% RSLogix 500 project aula1.RSS, saved by version 8.30.00.16 %
PROJECT "UNTITLED"    % processor: Bul.1763 MicroLogix 1100 Series B %

PROGRAM FILES
  LAD 2   6 rungs

DATA FILES
  O0 OUTPUT  4 elements
  I1 INPUT  6 elements
  S2 STATUS  66 elements
  B3 BINARY  1 elements
  T4 TIMER  1 elements
  C5 COUNTER  1 elements
  R6 CONTROL  1 elements
  N7 INTEGER  1 elements
  F8 FLOAT  1 elements

LADDER 2
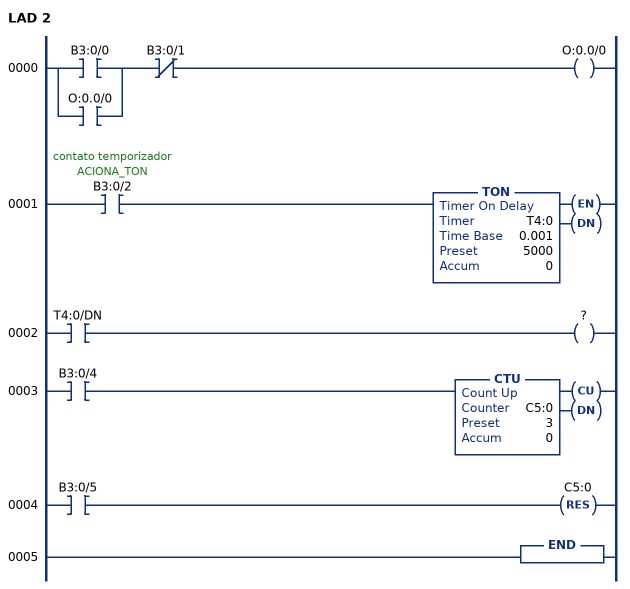
% Rung: 0 %
SOR BST XIC B3:0/0 NXB XIC O:0.0/0 BND XIO B3:0/1 OTE O:0.0/0 EOR
% Rung: 1 %  % edit flag set %
SOR XIC B3:0/2 TON T4:0 0.001 5000 0 EOR
%   B3:0/2  ACIONA_TON  "contato temporizador" %
% Rung: 2 %  % edit flag set %
SOR XIC T4:0/DN OTE ? EOR
% Rung: 3 %  % edit flag set %
SOR XIC B3:0/4 CTU C5:0 3 0 EOR
% Rung: 4 %  % edit flag set %
SOR XIC B3:0/5 RES C5:0 EOR
% Rung: 5 %
SOR END EOR
